PROGRAM ADSTesting
VAR
	fbAdsTest : ADSReadBasic;
	send: BOOL;
	Idx : UDINT := 16#01010010;
	off : UDINT := 16#00000010;
	results : UninTest;
END_VAR

IF send THEN
	fbAdsTest.SetADSReadTarget(TargetNetId := '127.0.0.1.1.1', 
							TargetPort := 351, 
							AdsIdxGrp := Idx, 
							AdsIdxOff := off, 
							ReadLength := 8, 
							ReadVarAddr  := ADR(results.resultArr));	
							
	fbAdsTest.Execute();
	IF fbAdsTest.Done THEN
		send := false;
	END_IF
END_IF
fbAdsTest();

END_PROGRAM

(* stored: Version 1.1.0.1, ProductVersion 3.1.4024.11
   POU ADSTesting: Id {d6b15b2b-a3b6-4245-8d86-1798190840d1}, SpecialFunc None *)
